Yaskawa INFORM job: R2_O3(0,-90)_AWOK.JBI

/JOB
//NAME R2_O3(0,-90)_AWOK
///FOLDERNAME PROGRAMY_TESTOWE_ODWLOK
//POS
///NPOS 33,33,33,2,0,0
///TOOL 0
///POSTYPE PULSE
///PULSE
C00000=-87506,26692,-6451,15797,58580,-60825
C00001=-86157,29655,-575,15266,56313,-60629
C00002=-85630,30926,1869,15063,55395,-60551
C00003=-84923,31899,2840,14605,55176,-60295
C00004=-85630,30926,1869,15063,55395,-60551
C00005=-86841,33013,5036,16034,54773,-61141
C00006=-86841,32894,6163,16181,54047,-61256
C00007=-86841,33013,5036,16034,54773,-61141
C00008=-73938,2382,-3106,-33786,21819,-37448
C00009=-73453,4428,3209,-39018,19717,-34959
C00010=-73972,6214,4746,-38205,19462,-35343
C00011=-73453,4428,3209,-39018,19717,-34959
C00012=-73938,2382,-3106,-33786,21819,-37448
C00013=-74377,7571,1351,-33183,21581,-37728
C00014=-74558,4812,-1726,-32244,21915,-38175
C00015=-75033,-1992,-9163,-30110,22670,-39191
C00016=-80432,-4266,-24752,15952,62758,-52954
C00017=-80434,-4257,-24745,15954,62759,-52955
C00018=-81259,-5326,-25609,16387,62901,-53249
C00019=-80434,-4143,-25899,15850,63499,-52849
C00020=-80434,-4257,-24745,15954,62759,-52955
C00021=-80434,-4257,-24745,15954,62759,-52955
C00022=-80434,-4257,-24745,15954,62759,-52955
C00023=-80432,-4266,-24752,15952,62758,-52954
C00024=-77087,-18045,-45485,6528,63632,-31215
C00025=-80448,-4218,-24714,11180,52424,-16549
C00026=-80446,-4219,-24714,11263,61777,-16174
C00027=-80082,-5585,-26617,11018,62189,-15996
C00028=-81271,-5287,-25577,11714,61874,-16475
C00029=-80447,-4219,-24714,14853,58765,-11509
C00030=-80456,-4194,-24694,16205,59267,-10401
C00031=-80452,-4208,-24705,20887,64890,-19794
C00032=-80452,-4208,-24705,17691,63208,-19920
BC00000=189887,628706,543657
BC00001=189887,628706,543657
BC00002=189887,628706,543657
BC00003=189887,628706,543657
BC00004=189887,628706,543657
BC00005=189887,628706,543657
BC00006=189887,628706,543657
BC00007=189887,628706,543657
BC00008=189887,628706,543657
BC00009=189887,628706,543657
BC00010=189887,628706,543657
BC00011=189887,628706,543657
BC00012=189887,628706,543657
BC00013=189887,628706,543657
BC00014=189887,628706,543657
BC00015=189887,628706,543657
BC00016=193928,682154,602974
BC00017=196175,682428,595414
BC00018=196175,682428,595414
BC00019=196175,682428,595414
BC00020=196185,687036,595495
BC00021=196200,694410,595624
BC00022=196210,699018,595705
BC00023=193962,698744,603266
BC00024=193919,675471,541467
BC00025=193880,654526,485848
BC00026=200662,667858,529060
BC00027=200662,667858,529060
BC00028=200662,667858,529060
BC00029=195157,662875,496351
BC00030=193857,647663,426077
BC00031=189076,659000,430993
BC00032=189873,652453,435399
EC00000=0,-556475
EC00001=0,-556475
EC00002=0,-556475
EC00003=0,-556475
EC00004=0,-556475
EC00005=0,-556475
EC00006=0,-556475
EC00007=0,-556475
EC00008=0,-556475
EC00009=0,-556475
EC00010=0,-556475
EC00011=0,-556475
EC00012=0,-556475
EC00013=0,-556475
EC00014=0,-556475
EC00015=0,-556475
EC00016=0,-556475
EC00017=0,-556475
EC00018=0,-556475
EC00019=0,-556475
EC00020=0,-556475
EC00021=0,-556475
EC00022=0,-556475
EC00023=0,-556475
EC00024=0,-556475
EC00025=0,-556475
EC00026=0,-556475
EC00027=0,-556475
EC00028=0,-556475
EC00029=0,-556475
EC00030=0,-556475
EC00031=0,-556475
EC00032=0,-556475
///POSTYPE BASE
///RECTAN
///RCONF 0,0,0,0,0,0,0,0,0,0,0,0,0,0,0,0,0,0,0,0,0,0,0,0
P00006=0.222,-3.123,-1.508,0.0000,0.0000,0.0000
P00021=-0.225,-6.128,-0.405,0.0000,0.0000,0.0000
//INST
///DATE 2023/11/22 16:22
///ATTR SC,RW
///GROUP1 RB1,BS1
///GROUP2 ST1
NOP
'r2_O3(0,-90
'Path S1195
SSFTOF
MOVJ C00000 BC00000 VJ=100.00  +MOVJ EC00000 VJ=100.00
MOVL C00001 BC00001 V=400.0  +MOVJ EC00001 VJ=100.00
SMOVL C00002 BC00002 V=60.0  +MOVJ EC00002
SREFP 3 C00003 BC00003  +REFP EC00003
CALL JOB:SEARCH-R1-S1
SET P021 P006
SSFTON P021
SMOVL C00004 BC00004 V=60.0  +MOVJ EC00004
SMOVL C00005 BC00005 V=60.0  +MOVJ EC00005
SREFP 3 C00006 BC00006  +REFP EC00006
CALL JOB:SEARCH-R1-S1
SET P021 P006
SSFTON P021
SMOVL C00007 BC00007 V=60.0  +MOVJ EC00007
SMOVL C00008 BC00008 V=100.0  +MOVJ EC00008
SMOVL C00009 BC00009 V=60.0  +MOVJ EC00009
SREFP 3 C00010 BC00010  +REFP EC00010
CALL JOB:SEARCH-R1-S1
SET P021 P006
SSFTON P021
SMOVL C00011 BC00011 V=60.0  +MOVJ EC00011
SMOVL C00012 BC00012 V=100.0  +MOVJ EC00012
SMOVL C00013 BC00013 V=100.0  +MOVJ EC00013
MOVL C00014 BC00014 V=400.0  +MOVJ EC00014 VJ=100.00
MOVL C00015 BC00015 V=1000.0  +MOVJ EC00015 VJ=100.00
'Path W1196
SSFTOF
SSFTON P021
SMOVL C00016 BC00016 V=400.0  +MOVJ EC00016
SMOVL C00017 BC00017 V=100.0 PL=0  +MOVJ EC00017
SREFP 1 C00018 BC00018  +REFP EC00018
SREFP 2 C00019 BC00019  +REFP EC00019
MACRO1 MJ#(0) ARGF0
ARCON
SMOVL C00020 BC00020 V=10.0  +MOVJ EC00020
SMOVL C00021 BC00021 V=10.0  +MOVJ EC00021
SMOVL C00022 BC00022 V=10.0  +MOVJ EC00022
ARCOF
SMOVL C00023 BC00023 V=400.0  +MOVJ EC00023
SSFTOF
'Path VIA1204
SSFTOF
MOVJ C00024 BC00024 VJ=100.00  +MOVJ EC00024 VJ=100.00
'Path W1197
SSFTOF
SSFTON P021
SMOVL C00025 BC00025 V=400.0  +MOVJ EC00025
SMOVL C00026 BC00026 V=100.0 PL=0  +MOVJ EC00026
SREFP 1 C00027 BC00027  +REFP EC00027
SREFP 2 C00028 BC00028  +REFP EC00028
MACRO1 MJ#(0) ARGF0
ARCON
SMOVL C00029 BC00029 V=10.0  +MOVJ EC00029
SMOVL C00030 BC00030 V=10.0  +MOVJ EC00030
SMOVL C00031 BC00031 V=10.0  +MOVJ EC00031
ARCOF
SMOVL C00032 BC00032 V=400.0  +MOVJ EC00032
SSFTOF
END
